(* CoDeSys 2.3.9.59 project: ProgettoSFC_NastroPistoneGiostra.pro *)
(* Libraries: STANDARD.LIB, Iecsfc.lib 12.5.98 12:03:00 *)

(* Task configuration *)
TASK Standard (PRIORITY := 0, INTERVAL := T#10ms);
	MAIN
END_TASK

(* Data type *)
TYPE ALTEZZA: (basso, alto);
END_TYPE

(* Data type *)
TYPE COLORE: (rosso, altro);
END_TYPE

(* Data type *)
TYPE PEZZO :
STRUCT
	Colore : COLORE;
	Altezza : ALTEZZA;
END_STRUCT
END_TYPE

(* Data type *)
TYPE POSTO :
STRUCT
	Presenza :BOOL:=FALSE;
	Pezzo :PEZZO;
	Ready :BOOL; (*uguale a 1 quando nel posto è terminato il lavoro*)
	Fine_Lavorazione :BOOL;
END_STRUCT
END_TYPE

(* POU MAIN, SFC *)
PROGRAM MAIN
VAR

(*Variabili Pistone*)
         (*Ingressi*)
	pezzo_magazzino  AT%IX0.0:BOOL;
	pistone_avanti AT%IX0.2:BOOL;
	pistone_indietro AT%IX0.4:BOOL;
         N_pezzi_spinti: INT:=0;
         (*Uscite*)
	pistone_on  AT%QX0.2:BOOL;
        (*TimerPistone*)
	timer_pistone: TON;
	mytime: TIME;
	timer_pist: BOOL:=TRUE;
	reset_timer: BOOL:=FALSE;

(*Variabili Nastro*)
         (*Ingressi*)
	fine_corsa_nastro  AT%IX0.6:BOOL;
         (*Uscite*)
	nastro_on  AT%QX0.0:BOOL;


(*Variabili Giostra*)
        Giostra: ARRAY[0..7] OF POSTO;
	i: INT :=0;
	j:INT:=0;
        (*Ingressi*)
        giostra_BUSY AT %IX6.1: BOOL;

        sensore_colore AT %IX2.1: BOOL;

        trapano_basso AT %IX2.5: BOOL ;
        trapano_alto AT %IX2.3: BOOL;

        tastatore_basso AT %IX5.3: BOOL;
        tastatore_alto AT %IX2.7: BOOL;

        pennarello_alto AT %IX5.4: BOOL;
        pennarello_basso AT %IX5.5: BOOL;

        pistone_PT5_avanti AT %IX5.0: BOOL;
        pistone_PT5_indietro AT %IX5.1: BOOL;

        pistone_PT6_avanti AT %IX5.7: BOOL;
        pistone_PT6_indietro AT %IX5.6: BOOL;

        pezzo_baia AT %IX5.2: BOOL;

        (*Uscite*)
        movimento_giostra AT %QX3.4: BOOL;

        trapano_on AT %QX3.7:BOOL;
        trapano_down AT %QX7.0: BOOL;

        tastatore_down AT %QX3.6: BOOL;

        pennarello_down AT %QX3.3: BOOL;

        pistone_PT5_on AT %QX3.1:BOOL ;
        pistone_PT6_on AT%QX3.5: BOOL;

	timer_giostra: BOOL;
	T_giostra: TON;
	mytimegiostra: TIME;
	T_trapano: TON;
	mytimetrapano: TIME;
	timer_trapano: BOOL;
END_VAR
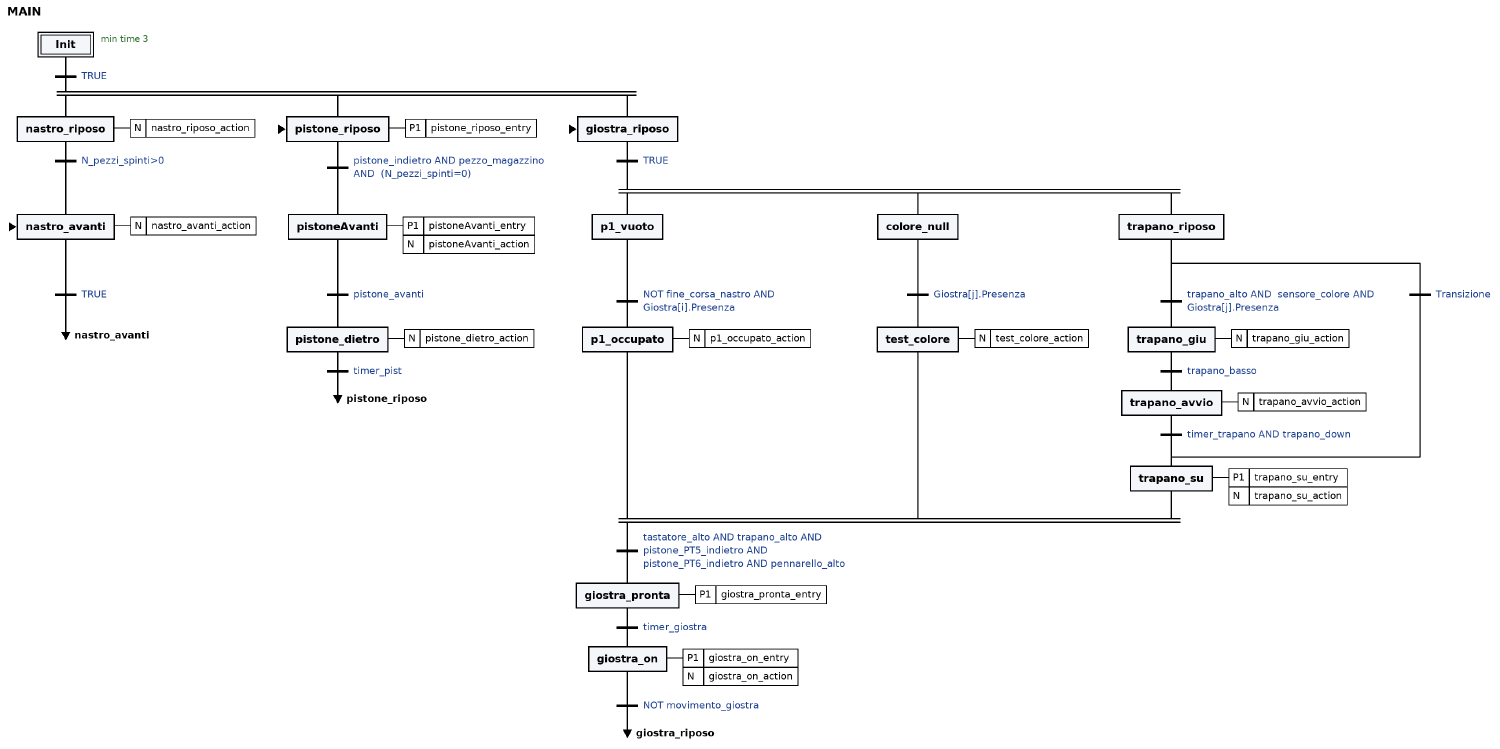
INITIAL_STEP Init: (* min time 3 *)
END_STEP
TRANSITION FROM Init TO (nastro_riposo, pistone_riposo, giostra_riposo) := TRUE;
END_TRANSITION
STEP nastro_riposo:
	nastro_riposo_action(N);
END_STEP
TRANSITION FROM nastro_riposo TO nastro_avanti := N_pezzi_spinti>0;
END_TRANSITION
STEP pistone_riposo:
	pistone_riposo_entry(P1);
END_STEP
TRANSITION FROM pistone_riposo TO pistoneAvanti := pistone_indietro AND pezzo_magazzino AND  (N_pezzi_spinti=0);
END_TRANSITION
STEP giostra_riposo:
END_STEP
TRANSITION FROM giostra_riposo TO (p1_vuoto, colore_null, trapano_riposo) := TRUE;
END_TRANSITION
STEP p1_vuoto:
END_STEP
TRANSITION FROM p1_vuoto TO p1_occupato := NOT fine_corsa_nastro AND Giostra[i].Presenza;
END_TRANSITION
STEP p1_occupato:
	p1_occupato_action(N);
END_STEP
STEP colore_null:
END_STEP
TRANSITION FROM colore_null TO test_colore := Giostra[j].Presenza;
END_TRANSITION
STEP test_colore:
	test_colore_action(N);
END_STEP
STEP trapano_riposo:
END_STEP
TRANSITION FROM trapano_riposo TO trapano_giu := trapano_alto AND  sensore_colore AND Giostra[j].Presenza;
END_TRANSITION
TRANSITION FROM trapano_riposo TO trapano_su := Transizione;
END_TRANSITION
STEP trapano_giu:
	trapano_giu_action(N);
END_STEP
TRANSITION FROM trapano_giu TO trapano_avvio := trapano_basso;
END_TRANSITION
STEP trapano_avvio:
	trapano_avvio_action(N);
END_STEP
TRANSITION FROM trapano_avvio TO trapano_su := timer_trapano AND trapano_down;
END_TRANSITION
STEP trapano_su:
	trapano_su_entry(P1);
	trapano_su_action(N);
END_STEP
TRANSITION FROM (p1_occupato, test_colore, trapano_su) TO giostra_pronta := tastatore_alto AND trapano_alto AND pistone_PT5_indietro AND pistone_PT6_indietro AND pennarello_alto;
END_TRANSITION
STEP giostra_pronta:
	giostra_pronta_entry(P1);
END_STEP
TRANSITION FROM giostra_pronta TO giostra_on := timer_giostra;
END_TRANSITION
STEP giostra_on:
	giostra_on_entry(P1);
	giostra_on_action(N);
END_STEP
TRANSITION FROM giostra_on TO giostra_riposo := NOT movimento_giostra;
END_TRANSITION
STEP pistoneAvanti:
	pistoneAvanti_entry(P1);
	pistoneAvanti_action(N);
END_STEP
TRANSITION FROM pistoneAvanti TO pistone_dietro := pistone_avanti;
END_TRANSITION
STEP pistone_dietro:
	pistone_dietro_action(N);
END_STEP
TRANSITION FROM pistone_dietro TO pistone_riposo := timer_pist;
END_TRANSITION
STEP nastro_avanti:
	nastro_avanti_action(N);
END_STEP
TRANSITION FROM nastro_avanti TO nastro_avanti := TRUE;
END_TRANSITION

ACTION nastro_riposo_action:
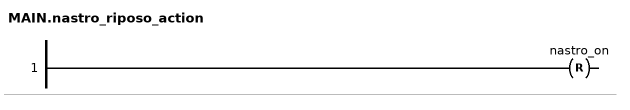
_LD_ (* Ladder Diagram *)
NETWORK 1
	* --- (R nastro_on)
_END_LD_
(* the same logic as Structured Text *)
(* Network 1 *)
nastro_on := FALSE;
END_ACTION

ACTION pistone_riposo_entry:
mytime:=t#0s;
END_ACTION

ACTION p1_occupato_action:
N_pezzi_spinti:=N_pezzi_spinti-1;
Giostra[i].Presenza:=TRUE;
i:=i+1;
END_ACTION

ACTION test_colore_action:
IF (sensore_colore=TRUE) THEN
Giostra[j].Pezzo.Colore:=rosso;
ELSE
Giostra[j].Pezzo.Colore:=altro;
END_IF
END_ACTION

ACTION trapano_giu_action:
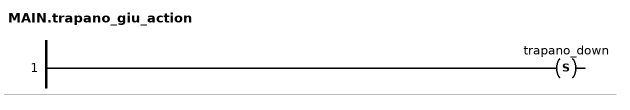
_LD_ (* Ladder Diagram *)
NETWORK 1
	* --- (S trapano_down)
_END_LD_
(* the same logic as Structured Text *)
(* Network 1 *)
trapano_down := TRUE;
END_ACTION

ACTION trapano_avvio_action:
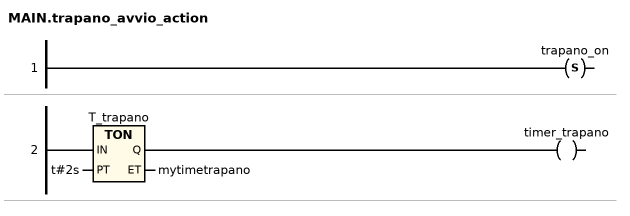
_LD_ (* Ladder Diagram *)
NETWORK 1
	* --- (S trapano_on)
NETWORK 2
	T_trapano:TON(IN: *, PT: t#2s, ET => mytimetrapano) --- (timer_trapano)
_END_LD_
(* the same logic as Structured Text *)
(* Network 1 *)
trapano_on := TRUE;
(* Network 2 *)
T_trapano(IN := TRUE, PT := t#2s);
mytimetrapano := T_trapano.ET;
timer_trapano := T_trapano.Q;
END_ACTION

ACTION trapano_su_entry:
mytimetrapano:=t#0s;
END_ACTION

ACTION trapano_su_action:
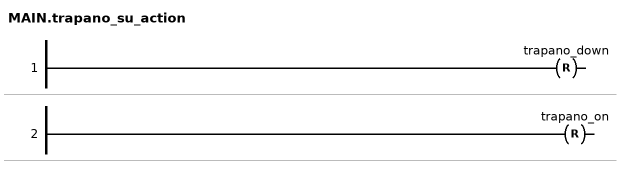
_LD_ (* Ladder Diagram *)
NETWORK 1
	* --- (R trapano_down)
NETWORK 2
	* --- (R trapano_on)
_END_LD_
(* the same logic as Structured Text *)
(* Network 1 *)
trapano_down := FALSE;
(* Network 2 *)
trapano_on := FALSE;
END_ACTION

ACTION giostra_pronta_entry:
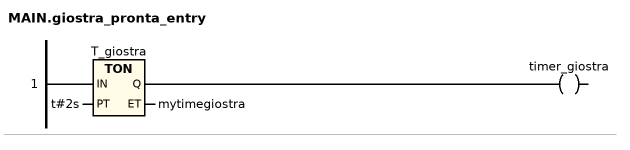
_LD_ (* Ladder Diagram *)
NETWORK 1
	T_giostra:TON(IN: *, PT: t#2s, ET => mytimegiostra) --- (timer_giostra)
_END_LD_
(* the same logic as Structured Text *)
(* Network 1 *)
T_giostra(IN := TRUE, PT := t#2s);
mytimegiostra := T_giostra.ET;
timer_giostra := T_giostra.Q;
END_ACTION

ACTION giostra_on_entry:
mytimegiostra:=t#0s;
j:=j+1;
END_ACTION

ACTION giostra_on_action:
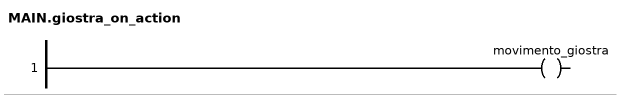
_LD_ (* Ladder Diagram *)
NETWORK 1
	* --- (movimento_giostra)
_END_LD_
(* the same logic as Structured Text *)
(* Network 1 *)
movimento_giostra := TRUE;
END_ACTION

ACTION pistoneAvanti_entry:
N_pezzi_spinti:=N_pezzi_spinti+1;
END_ACTION

ACTION pistoneAvanti_action:
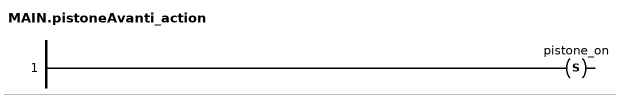
_LD_ (* Ladder Diagram *)
NETWORK 1
	* --- (S pistone_on)
_END_LD_
(* the same logic as Structured Text *)
(* Network 1 *)
pistone_on := TRUE;
END_ACTION

ACTION pistone_dietro_action:
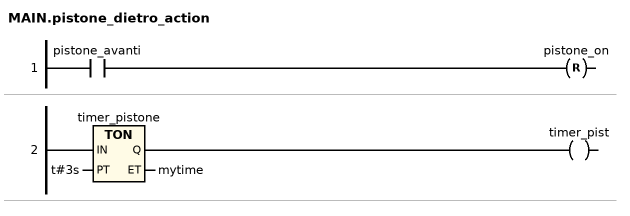
_LD_ (* Ladder Diagram *)
NETWORK 1
	[pistone_avanti] --- (R pistone_on)
NETWORK 2
	timer_pistone:TON(IN: *, PT: t#3s, ET => mytime) --- (timer_pist)
_END_LD_
(* the same logic as Structured Text *)
(* Network 1 *)
IF pistone_avanti THEN pistone_on := FALSE; END_IF;
(* Network 2 *)
timer_pistone(IN := TRUE, PT := t#3s);
mytime := timer_pistone.ET;
timer_pist := timer_pistone.Q;
END_ACTION

ACTION nastro_avanti_action:
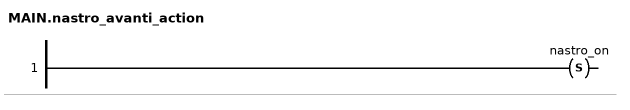
_LD_ (* Ladder Diagram *)
NETWORK 1
	* --- (S nastro_on)
_END_LD_
(* the same logic as Structured Text *)
(* Network 1 *)
nastro_on := TRUE;
END_ACTION

TRANSITION Transizione:
trapano_alto AND (NOT sensore_colore OR Giostra[i].Presenza=FALSE)
END_TRANSITION
END_PROGRAM
